PROGRAM MAIN
VAR	
	Control : FB2_Control;
	Modules : FB3_Modules;
	
END_VAR

Control();
Modules();

END_PROGRAM

(* stored: Version 1.1.0.1, ProductVersion 3.1.4024.6
   POU MAIN: Id {3bcc1047-ddf4-456f-8ab1-83140f54896c}, SpecialFunc None *)
